PROGRAM MAIN
VAR	
END_VAR

StateProgram();

END_PROGRAM

(* stored: Version 1.1.0.1, ProductVersion 3.1.4024.12
   POU MAIN: Id {0ce4d6ef-3580-40cb-80fe-c304716bd060}, SpecialFunc None *)
